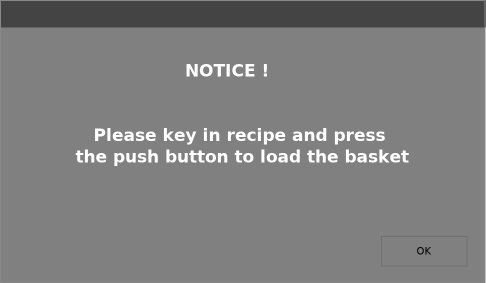
VISUALIZATION Popup_Ld_Warning  // 486x283
    Rectangle (0,0 485x283)
    Rectangle (1,0 485x27)
    Label (152,51 151x39), "NOTICE !"
    Label (10,78 465x136), "Please key in recipe and press the push button to load the basket"
    Button (381,236 86x30), "OK", colour toggle: bPopupPageRapidConfirm
        tap bPopupPageRapidConfirm
END_VISUALIZATION

(* stored: Version 1.1.0.1, ProductVersion 3.1.4024.12
   Visu Popup_Ld_Warning: Id {1dc05103-0fe9-4102-baae-70e86a9d7483} *)
